{attribute 'qualified_only' := ''}
TYPE E_Mode :
(
	INITIALIZED := 0,
	AUTO := 10,
	SEMI := 11,
	MANU := 12
);
END_TYPE

(* stored: Version 1.1.0.1, ProductVersion 3.1.0.14
   DUT E_Mode: Id {2cc6d00b-d8f0-426c-9ff2-97a490f63eb9} *)
